Universal Robots PolyScope program: RC_E1_MOVE_110.urp

Program RC_E1_MOVE_110 (createdIn=3.0.0 lastSavedIn=3.0.0 directory=/programs installation=default)
Robot Program (runOnlyOnce=true motionType=MoveJ speed=1.047198 acceleration=1.396263 useActiveTCP=false)
  'Program generated by RoboDK v4.1.0 for UR3e_HORNO on 05/09/2022 13:21:51'
  'Using nominal kinematics.'
  'Using Ref. UR3_2: p[0.000000, 0.000000, 0.000000, 0.000000, 0.000000, 0.000000]'
  'Using TCP 0208-0001-0001-307-000-3 Horno: p[0.000000, 0.000000, 0.164750, 0.000000, 0.000000, 0.000000]'
  Script: set_tcp(p[0.000000, 0.000000, 0.164750, 0.000000, 0.000000, 0.000000])
  Script: movej([0.200016, -1.409861, -0.955490, -2.344949, 1.570623, 0.000002],0.60000,0.12500,0,0.0000)
